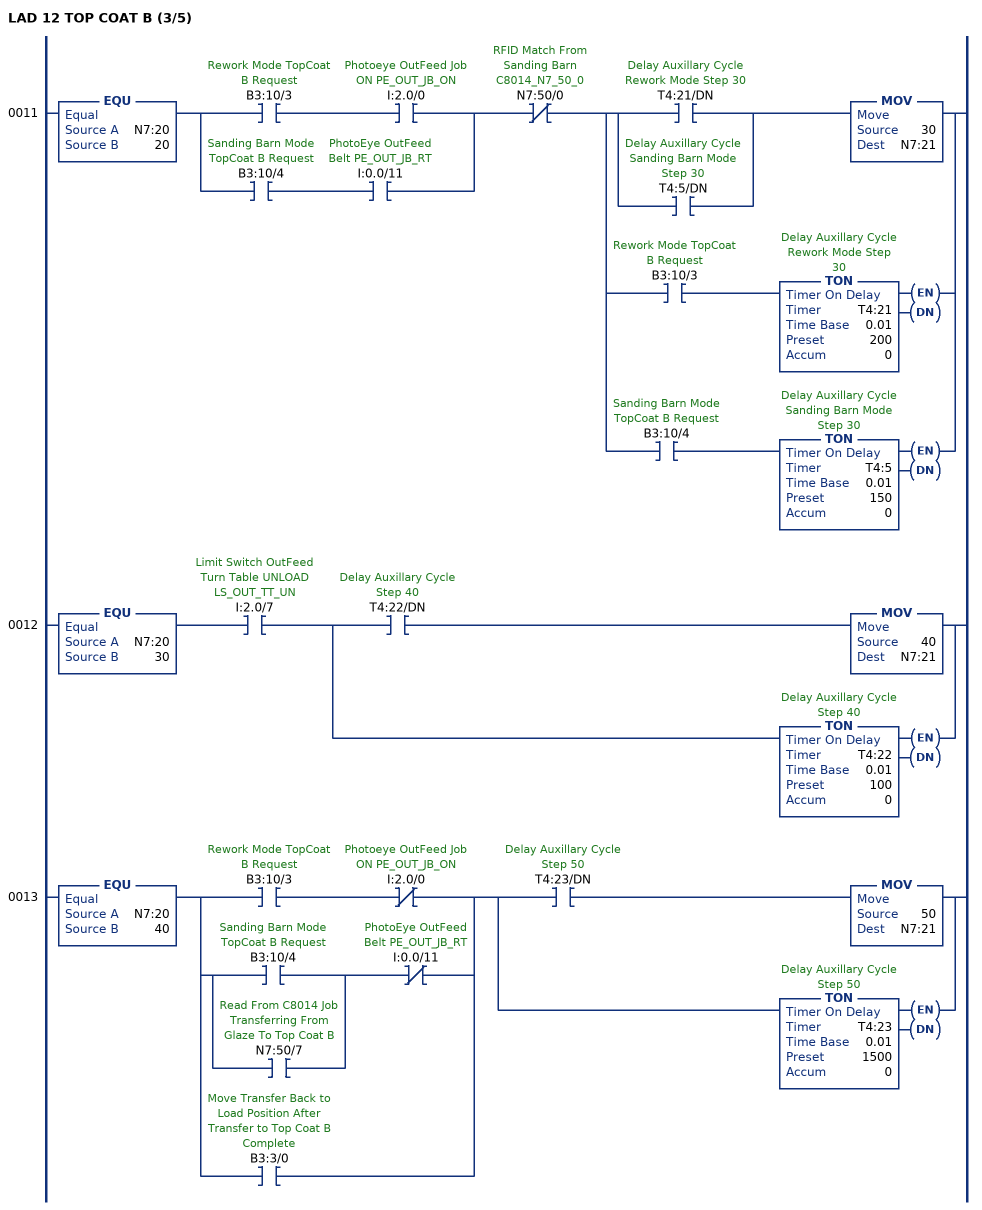
% Rung: 11 %
SOR EQU N7:20 20 BST XIC B3:10/3 XIC I:2.0/0 NXB XIC B3:10/4 XIC I:0.0/11 BND XIO N7:50/0 BST BST XIC T4:21/DN NXB XIC T4:5/DN BND MOV 30 N7:21 NXB XIC B3:10/3 TON T4:21 0.01 200 0 NXB XIC B3:10/4 TON T4:5 0.01 150 0 BND EOR
%   B3:10/3  "Rework Mode TopCoat B Request" %
%   I:2.0/0  PE_OUT_JB_ON  "Photoeye OutFeed Job ON" %
%   B3:10/4  "Sanding Barn Mode TopCoat B Request" %
%   I:0.0/11  PE_OUT_JB_RT  "PhotoEye OutFeed Belt" %
%   N7:50/0  C8014_N7_50_0  "RFID Match From Sanding Barn" %
%   T4:21  "Delay Auxillary Cycle Rework Mode Step 30" %
%   T4:5  "Delay Auxillary Cycle Sanding Barn Mode Step 30" %
% Rung: 12 %
SOR EQU N7:20 30 XIC I:2.0/7 BST XIC T4:22/DN MOV 40 N7:21 NXB TON T4:22 0.01 100 0 BND EOR
%   I:2.0/7  LS_OUT_TT_UN  "Limit Switch OutFeed Turn Table UNLOAD" %
%   T4:22  "Delay Auxillary Cycle Step 40" %
% Rung: 13 %
SOR EQU N7:20 40 BST XIC B3:10/3 XIO I:2.0/0 NXB BST XIC B3:10/4 NXB XIC N7:50/7 BND XIO I:0.0/11 NXB XIC B3:3/0 BND BST XIC T4:23/DN MOV 50 N7:21 NXB TON T4:23 0.01 1500 0 BND EOR
%   B3:10/3  "Rework Mode TopCoat B Request" %
%   I:2.0/0  PE_OUT_JB_ON  "Photoeye OutFeed Job ON" %
%   B3:10/4  "Sanding Barn Mode TopCoat B Request" %
%   N7:50/7  "Read From C8014 Job Transferring From Glaze To Top Coat B" %
%   I:0.0/11  PE_OUT_JB_RT  "PhotoEye OutFeed Belt" %
%   B3:3/0  "Move Transfer Back to Load Position After Transfer to Top Coat B Complete" %
%   T4:23  "Delay Auxillary Cycle Step 50" %

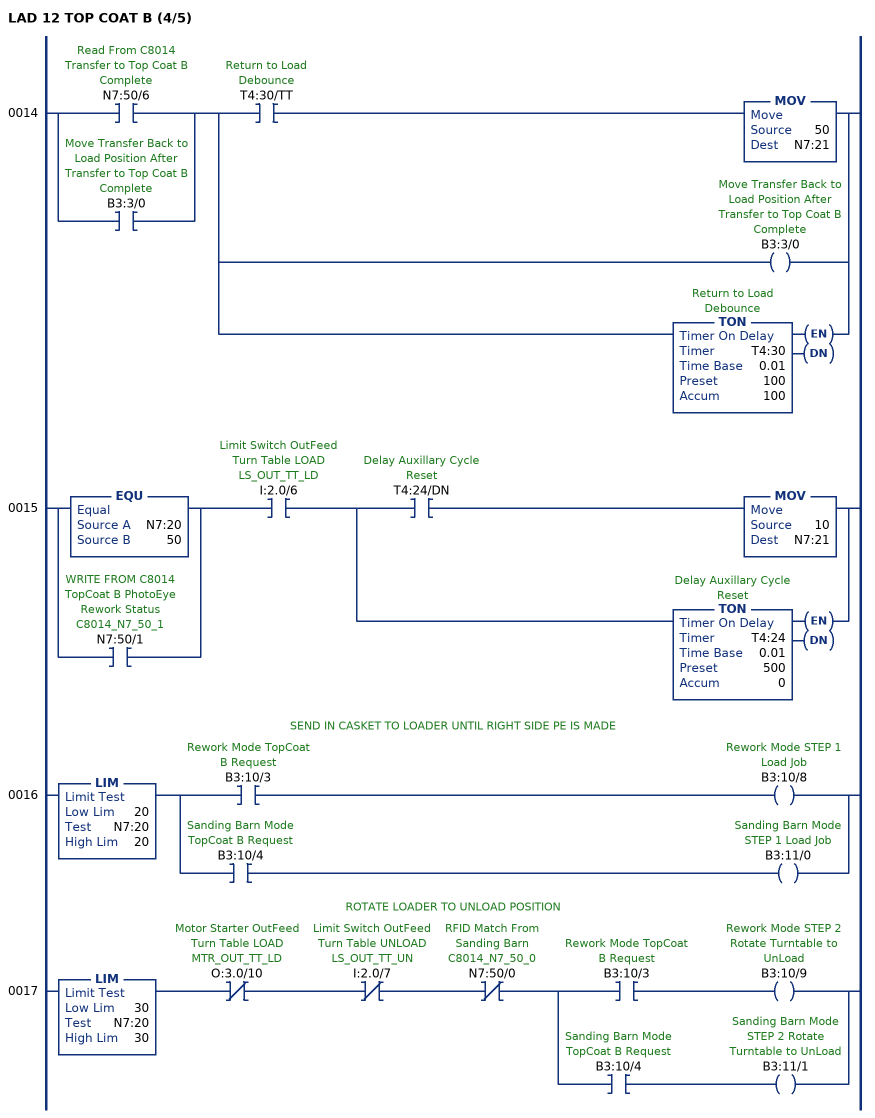
% Rung: 14 %
SOR BST XIC N7:50/6 NXB XIC B3:3/0 BND BST XIC T4:30/TT MOV 50 N7:21 NXB OTE B3:3/0 NXB TON T4:30 0.01 100 100 BND EOR
%   N7:50/6  "Read From C8014 Transfer to Top Coat B Complete" %
%   B3:3/0  "Move Transfer Back to Load Position After Transfer to Top Coat B Complete" %
%   T4:30  "Return to Load Debounce" %
% Rung: 15 %
SOR BST EQU N7:20 50 NXB XIC N7:50/1 BND XIC I:2.0/6 BST XIC T4:24/DN MOV 10 N7:21 NXB TON T4:24 0.01 500 0 BND EOR
%   N7:50/1  C8014_N7_50_1  "WRITE FROM C8014 TopCoat B PhotoEye Rework Status" %
%   I:2.0/6  LS_OUT_TT_LD  "Limit Switch OutFeed Turn Table LOAD" %
%   T4:24  "Delay Auxillary Cycle Reset" %
% Rung: 16 %
% SEND IN CASKET TO LOADER UNTIL RIGHT SIDE PE IS MADE %
SOR LIM 20 N7:20 20 BST XIC B3:10/3 OTE B3:10/8 NXB XIC B3:10/4 OTE B3:11/0 BND EOR
%   B3:10/3  "Rework Mode TopCoat B Request" %
%   B3:10/8  "Rework Mode STEP 1 Load Job" %
%   B3:10/4  "Sanding Barn Mode TopCoat B Request" %
%   B3:11/0  "Sanding Barn Mode STEP 1 Load Job" %
% Rung: 17 %
% ROTATE LOADER TO UNLOAD POSITION %
SOR LIM 30 N7:20 30 XIO O:3.0/10 XIO I:2.0/7 XIO N7:50/0 BST XIC B3:10/3 OTE B3:10/9 NXB XIC B3:10/4 OTE B3:11/1 BND EOR
%   O:3.0/10  MTR_OUT_TT_LD  "Motor Starter OutFeed Turn Table LOAD" %
%   I:2.0/7  LS_OUT_TT_UN  "Limit Switch OutFeed Turn Table UNLOAD" %
%   N7:50/0  C8014_N7_50_0  "RFID Match From Sanding Barn" %
%   B3:10/3  "Rework Mode TopCoat B Request" %
%   B3:10/9  "Rework Mode STEP 2 Rotate Turntable to UnLoad" %
%   B3:10/4  "Sanding Barn Mode TopCoat B Request" %
%   B3:11/1  "Sanding Barn Mode STEP 2 Rotate Turntable to UnLoad" %

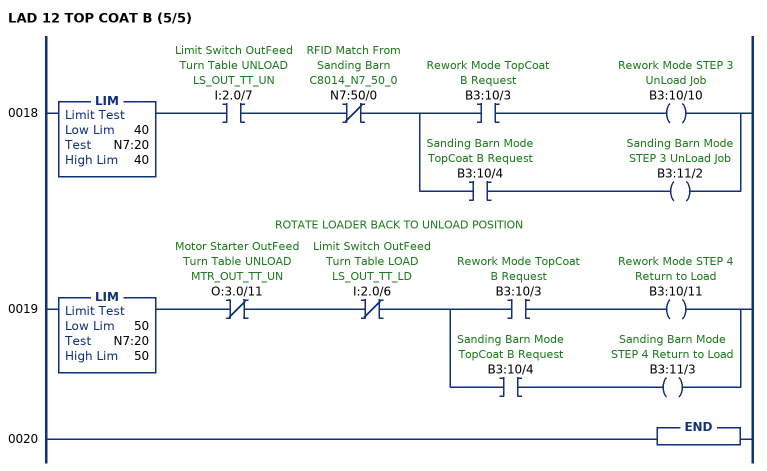
% Rung: 18 %
SOR LIM 40 N7:20 40 XIC I:2.0/7 XIO N7:50/0 BST XIC B3:10/3 OTE B3:10/10 NXB XIC B3:10/4 OTE B3:11/2 BND EOR
%   I:2.0/7  LS_OUT_TT_UN  "Limit Switch OutFeed Turn Table UNLOAD" %
%   N7:50/0  C8014_N7_50_0  "RFID Match From Sanding Barn" %
%   B3:10/3  "Rework Mode TopCoat B Request" %
%   B3:10/10  "Rework Mode STEP 3 UnLoad Job" %
%   B3:10/4  "Sanding Barn Mode TopCoat B Request" %
%   B3:11/2  "Sanding Barn Mode STEP 3 UnLoad Job" %
% Rung: 19 %
% ROTATE LOADER BACK TO UNLOAD POSITION %
SOR LIM 50 N7:20 50 XIO O:3.0/11 XIO I:2.0/6 BST XIC B3:10/3 OTE B3:10/11 NXB XIC B3:10/4 OTE B3:11/3 BND EOR
%   O:3.0/11  MTR_OUT_TT_UN  "Motor Starter OutFeed Turn Table UNLOAD" %
%   I:2.0/6  LS_OUT_TT_LD  "Limit Switch OutFeed Turn Table LOAD" %
%   B3:10/3  "Rework Mode TopCoat B Request" %
%   B3:10/11  "Rework Mode STEP 4 Return to Load" %
%   B3:10/4  "Sanding Barn Mode TopCoat B Request" %
%   B3:11/3  "Sanding Barn Mode STEP 4 Return to Load" %
% Rung: 20 %
SOR END EOR

OTHER DOCUMENTED ADDRESSES
  B3:0/14  RST_EN
  B3:2  "LaneSelection"
  B3:5/8  INF_CYC_8  "InFeed Cycle Transfer Down"
  B3:6/0  "MAN Selector SW FWD"
  B3:6/1  "MAN Selector SW REV"
  B3:7/0  POS_MAP_OUT_CAM_1  "Position Map Cam 1 OutFeed"
  B3:7/1  POS_MAP_OUT_CAM_2  "Position Map Cam 2 Slow Speed OutFeed"
  B3:7/2  POS_MAP_OUT_CAM_3  "Position Map Cam 3 OutFeed"
  B3:18/0  POS_OMAP_CAM_1  "Position Map Cam 1 OutFeed"
  B9:5/14  INF_SLO_SPD  "InFeed Slow Speed"
  B9:8/0  OUT_BOT_LD  "OutFeed Botom Load"
  B9:8/1  OUT_TOP_LD  "OutFeed Top Load"
  B9:8/13  OUT_HLD_UN  "OutFeed Hold Load"
  B9:8/14  OUT_SLO_SPD  "OutFeed Slow Speed"
  I:0.0/12  BELT_LEFT_END_PE
  I:1.0/7  "Spare"
  I:4.0/0  PR_OUT_CAM_1  "Proximity Switch OutFeed Cam 1"
  I:4.0/1  PR_OUT_CAM_2  "Proximity Switch OutFeed Cam 2"
  I:4.0/2  PR_OUT_CAM_3  "Proximity Switch OutFeed Cam 3"
  I:4.0/3  FS_OUT_1  "Foot Switch OutFeed Lane 1"
  I:4.0/4  FS_OUT_2  "Foot Switch OutFeed Lane 2"
  I:4.0/5  FS_OUT_3  "Foot Switch OutFeed Lane 3"
  I:4.0/6  "Spare"
  I:4.0/7  PB_RST_LN  "Spare"
  MG11:0  "Read N7:51 from M8014"
  MG11:1  "Write N7:5 TO C8014"
  MG11:2  "READ FROM M8017 N7:0 TO N7:10"
  MG11:3  "Write N7:51 TO M8017"
  N7:1/15  C8011_N7_5_15  "Writing From C8011 TopCoat A Heartbeat Pulse"
  N7:4  INF_CSP  "InFeed Current Section Posi"
  N7:5/0  "N7:5 Write to M8014 C is running"
  N7:7  _OUT_CSP  "OutFeed Current Section Posi"
  N7:10/0  "Lane(1) Position Data"
  N7:10/1  "Lane (2) Position Data"
  N7:10/2  "Lane (3) Position Data"
  N7:10/3  "Lane (3) Position Data"
  N7:14  INF_NSP  "InFeed Next Section Positio"
  N7:17  OUT_NSP  "OutFeed Next Section Positio"
  N7:40  INF_FIFO_DEST  "InFeed FIFO Destination"
  N7:41  INF_FIFO_1  "InFeed FIFO Buffer Position 1"
  N7:42  INF_FIFO_2  "InFeed FIFO Buffer Position 2"
  N7:43  INF_FIFO_3  "InFeed FIFO Buffer Position 3"
  N7:44  INF_FIFO_4  "InFeed FIFO Buffer Position 4"
  N7:73  OUT_FIFO_3  "OutFeed FIFO Buffer Position 3"
  N7:74  OUT_FIFO_4  "OutFeed FIFO Buffer Position 4"
  N7:75  OUT_FIFO_5  "OutFeed FIFO Buffer Position 5"
  N7:76  OUT_FIFO_6  "OutFeed FIFO Buffer Position 6"
  N7:77  OUT_FIFO_7  "OutFeed FIFO Buffer Position 7"
  N7:78  OUT_FIFO_8  "OutFeed FIFO Buffer Position 8"
  N71:40  INF_FIFO_POL_DEST  "InFeed FIFO Polish Buffer Destination"
  N71:41  INF_FIFO_POL_1  "InFeed FIFO Polish Buffer Position 1"
  N71:42  INF_FIFO_POL_2  "InFeed FIFO Polish Buffer Position 2"
  N71:43  INF_FIFO_POL_3  "InFeed FIFO Polish Buffer Position 3"
  N71:44  INF_FIFO_POL_4  "InFeed FIFO Polish Buffer Position 4"
  N71:45  INF_FIFO_POL_5  "InFeed FIFO Polish Buffer Position 5"
  N71:46  INF_FIFO_POL_6  "InFeed FIFO Polish Buffer Position 6"
  N71:47  INF_FIFO_POL_7  "InFeed FIFO Polish Buffer Position 7"
  N71:48  INF_FIFO_POL_8  "InFeed FIFO Polish Buffer Position 8"
  N71:70  OUT_FIFO_STA_DEST  "OutFeed FIFO Sanding Station Destination"
  N71:71  OUT_FIFO_STA_1  "OutFeed FIFO Sanding Station Position 1"
  N71:72  OUT_FIFO_STA_2  "OutFeed FIFO Sanding Station Position 2"
  N71:73  OUT_FIFO_STA_3  "OutFeed FIFO Sanding Station Position 3"
  NEQ  
  O  
  O:0.0/3  MTR_OUT_TRAV_FWD  "Motor Starter OutFeed Travel Forward"
  O:0.0/4  MTR_OUT_TRAV_REV  "Motor Starter OutFeed Travel Reverse"
  O:0.0/5  MTR_OUT_TRAV_FST  "Motor Starter OutFeed Travel Fast"
  O:2.0/0  "InfeedRaiseMotor"
  O:2.0/1  "OutfeedRaiseMotor"
  O:2.0/2  "UpperOvenSolenoid"
  O:2.0/3  "UpperOvenChain"
  O:2.0/4  "InfeedLowerMotor"
  O:2.0/5  "OutputLowerMotor"
  O:3.0/2  "Spare"
  O:3.0/3  "Spare"
  O:3.0/5  SOL_IN_RE  "Solenoid InFeed Arms Retract"
  O:3.0/13  SOL_OUT_RE  "Solenoid OutFeed Arms Retract"
  PE2_ZONE_A  
  T4:7  "RotateDelayTimer"
  T4:8  "TIME DELAY TO MAKE SURE CASKET IS OUT OF THE LOADER"
  T4:9  "RotateTableDelay"
  T4:13/TT  "Unload Black Belt Conveyor"
  T4:40  TMR_INF_DLY_POS_UD  "Timer InFeed Delay Position Updat"
  T4:50  TMR_INF_DBN_CYC_0  "Timer InFeed Debounce Cycle 0"
  T4:59  TMR_INF_DBN_CYC_9  "Timer InFeed Debounce Cycle 9"
  T4:64  TMR_LN_5  "Timer Lane 5 RunTime"
  T4:66  TMR_LN_6  "Timer Lane 6 RunTime"
  T4:67  TMR_LN_7  "Timer Lane 7 RunTime"
  T4:68  TMR_LN_8  "Timer Lane 8 RunTime"
  T4:70  TMR_OUT_DLY_POS_UD  "Timer OutFeed Delay Position Updat"
  T4:80  TMR_OUT_DBN_CYC_0  "Timer OutFeed Debounce Cycle 0"
  T9:0  "DebounceTimer1"
  T9:4  "DebounceTimer5"
  T9:5  "AirbagDownDelay"
  T9:6  "AirbagDownTimer"
  T9:7  "AirbagsDownTimer"
  T9:8  "AirbagsDownTimer"
  T9:12  "Delay Integer Update"
  T9:13  "Home Position Debounce"
  T9:15  "Update Integer Debounce"
  T9:15/DN  "IntegerUpdate Debounce"
  T9:18  "Delay N7:30 Zero"
  T20:0  "DebounceTimer1"
  T41:62  TMR_DBN_FFL_LN_3  "Timer Debounce Lane 3"
  T41:63  TMR_DBN_FFL_LN_4  "Timer Debounce Lane 4"
  T41:64  TMR_DBN_FFL_LN_5  "Timer Debounce Lane 5"
  T41:65  TMR_DBN_FFL_LN_6  "Timer Debounce Lane 6"
  T41:66  TMR_DBN_FFL_LN_7  "Timer Debounce Lane 7"
  T41:67  TMR_DBN_FFL_LN_8  "Timer Debounce Lane 8"

COMMENTS NOT ATTACHED TO A CURRENT RUNG
  U:3: Jump to Load Lower Belt
  N7:30: Lane Select Logic
  T4:10: UNLOADE CASKET TO TOPCOAT B
  B3:10/11: STEP 4 ROTATE LOADER BACK TO LOAD POSITION
  T4:8: STEP 3 SEND CASKET TO TOPCOAT B
  B3:10/9: STEP 2 ROTATE TO UNLOAD POSITION
  B3:10/8: STEP 1 SEND CASKET TO LOADER UNTIL LEFT SIDE PHOTO EYE
  B3:10/7: SANDING BARN CYCLE MODE
  N7:5/0: Telling C8014 When Oven B is running

DATA TABLE (non-zero values as saved)
DATA B3
% B3:0 % 0X2A80 0X0000 0X0000 0X0001 0X0000 0X0100 0X0000 0X0005 0X0200 0X0000
% B3:10 % 0X0040 0X0000 0X0000 0X0000 0X0000 0X0000 0X0000 0X0000 0X0000 0X0000
DATA T4
% .PRE .ACC %
% T4:0 % 300 0
% T4:1 % 75 0
% T4:2 % 50 0
% T4:3 % 50 0
% T4:4 % 262 215
% T4:5 % 150 0
% T4:6 % 100 0
% T4:7 % 2 2
% T4:8 % 200 0
% T4:9 % 2 0
% T4:10 % 200 0
% T4:11 % 120 0
% T4:12 % 2 0
% T4:13 % 800 0
% T4:14 % 2 0
% T4:15 % 200 0
% T4:16 % 5 0
% T4:20 % 200 0
% T4:21 % 200 0
% T4:22 % 100 0
% T4:23 % 1500 0
% T4:24 % 500 0
% T4:30 % 100 100
% T4:51 % 10 0
% T4:52 % 75 0
% T4:53 % 10 0
% T4:54 % 200 0
% T4:55 % 100 0
% T4:56 % 200 0
% T4:57 % 200 0
% T4:58 % 200 0
% T4:60 % 60 34
% T4:61 % 60 17
% T4:62 % 524 0
% T4:63 % 524 0
% T4:70 % 100 0
% T4:81 % 200 0
% T4:82 % 200 0
% T4:83 % 200 0
% T4:84 % 200 0
% T4:85 % 200 69
% T4:86 % 5 0
% T4:87 % 200 0
% T4:88 % 1000 0
% T4:89 % 200 0
DATA C5
% .PRE .ACC %
% C5:1 % 10000 0
% C5:4 % 0 13325
% C5:5 % 0 10354
DATA R6
% .LEN .POS %
% R6:0 % 8 0
% R6:3 % 9 0
% R6:4 % 2 1
% R6:5 % 3 0
DATA N7
% N7:0 % 0 0 0 0 0 0 0 5 0 0
% N7:20 % 20 10 0 0 0 0 0 0 0 0
% N7:50 % 8 0 0 0 0 0 0 0 0 0
% N7:60 % 1 0 0 0 0 0 0 0 0 0
% N7:70 % 2 2 0 0 0 0 0 0 0 0
DATA B9
% B9:0 % 0X0002 0X0000 0X0000 0X0000 0X0000 0X0000 0X0002 0X0000 0X0800 0X0000
DATA B10
% B10:0 % 0X0000 0X0000 0X0000 0X0000 0X0000 0X0000 0X0000 0X0000 0X0003 0X0000
DATA T41
% .PRE .ACC %
% T41:60 % 500 0
% T41:61 % 500 500
